{attribute 'GeneratedUsingTerminal: EL2622-0000-0016'}
{attribute addProperty BoxType "EL2622-0000-0016"}
{attribute addProperty Description "EL2622 2Ch. Relay Output, NO (230V AC / 30V DC)"}
{attribute addProperty Physics "KK"}
{attribute addProperty Id "Channel_1AT %Q*Channel_42CA91F71Channel_2AT %Q*Channel_42CA91F71WcStateAT %I*WcState_0B2B16F91InfoDataAT %I*InfoData_6F19DB2B2"}
{attribute addProperty CRC "2954971456"}
{attribute addProperty Size "5"}
TYPE EL2622_B0214940 EXTENDS EtcSlaveTerminalBase_947E5A46 :
STRUCT
	{attribute addProperty Name "Channel_1"}
	Channel_1 : Channel_42CA91F7;
	{attribute addProperty Name "Channel_2"}
	Channel_2 : Channel_42CA91F7;
	{attribute addProperty Name "WcState"}
	WcState : WcState_0B2B16F9;
	{attribute addProperty Name "InfoData"}
	InfoData : InfoData_6F19DB2B;
END_STRUCT
END_TYPE

(* stored: Version 1.2.0.0, ProductVersion 3.1.4024.11
   DUT EL2622_B0214940: Id {db22b4c9-da3a-4f6a-914b-3c5dcb2cb957} *)
